Fanuc KAREL source: kx00008.KL

-- PROVISIONAL review KL for V940-1; original PC SHA256 1ecd864a25350347dfaac4f31079a7991ab00b4250fa72b735314c4ba797eecd
-- Incomplete behavior may be omitted. Consult companion uncertainty JSON. Do not deploy.
PROGRAM KX00008
%NOLOCKGROUP
VAR
  I : INTEGER
  J : INTEGER
  B : BOOLEAN
  F : FILE
  S : STRING[80]
-- UNRESOLVED_DECL P type=000102
BEGIN
  -- V9_ZERO_TABLE_METADATA_HINT layout=0001; no indexed target words; source/name/runtime held
  -- UNRESOLVED_PC offsets 5-7; opcodes 9C,3A
  -- UNRESOLVED_PC offsets 12-16; opcodes 7F
END KX00008
